{attribute 'linkalways'} 
{attribute 'no_explicit_call' := 'This FB is a CLASS and must be accessed using methods or properties'}
{attribute 'enable_dynamic_creation'}
FUNCTION_BLOCK _Array0to1OfARRAYTYP EXTENDS ArrayDatatypeBase
VAR CONSTANT
	lBound : DINT := 0;
	uBound : DINT := 1;
END_VAR
VAR
	localData : ARRAY [lBound..uBound] OF ARRAYTYP;
	activeData : REFERENCE TO ARRAY [lBound..uBound] OF ARRAYTYP REF= localData;
	elements : ARRAY [lBound..uBound] OF _ARRAYTYP();
	baseType : _ARRAYTYP();
END_VAR

PROPERTY PUBLIC Address : PVOID
GET
Address := ADR(activeData);
END_GET
END_PROPERTY

PROPERTY PUBLIC BaseDatatype : I_Datatype
GET
BaseDatatype := baseType;
END_GET
END_PROPERTY

METHOD PUBLIC ClearReference
VAR_INPUT
END_VAR
activeData REF= localData;
SetElementReference();
END_METHOD

METHOD PUBLIC Clone : I_Datatype
VAR
    pClone : POINTER TO _;
END_VAR
pClone := __NEW(_());
pClone^.Value := Value;
Clone := pClone^;
END_METHOD

METHOD FB_init : BOOL
VAR_INPUT
	bInitRetains : BOOL; // if TRUE, the retain variables are initialized (warm start / cold start)
	bInCopyCode : BOOL;  // if TRUE, the instance afterwards gets moved into the copy code (online change)
END_VAR
SetElementReference();
END_METHOD

METHOD PUBLIC GetElementAsDatatypeByIndex : I_Datatype
VAR_INPUT
	Index : DINT;
END_VAR
GetElementAsDatatypeByIndex := elements[Index];
END_METHOD

METHOD PUBLIC GetElementByIndex : REFERENCE TO _ARRAYTYP;
VAR_INPUT
	Index : DINT;
END_VAR
GetElementByIndex REF= elements[Index];
END_METHOD

PROPERTY PUBLIC LowerBound : DINT
GET
LowerBound := lBound;
END_GET
END_PROPERTY

METHOD PUBLIC MakeReferenceTo
VAR_INPUT
	ReferenceTarget : REFERENCE TO ARRAY [lBound..uBound] OF ARRAYTYP;
END_VAR
activeData REF= ReferenceTarget;
SetElementReference();
END_METHOD

METHOD PROTECTED OnSerializeArrayValues
VAR_INPUT
	Serializer : I_Serializer;
END_VAR
VAR
	i : DINT;
END_VAR
FOR i := lBound TO uBound DO
	elements[i].SerializeWith(Serializer);
END_FOR
END_METHOD

METHOD PROTECTED SetElementReference
VAR_INPUT
END_VAR
VAR
	i : DINT;
END_VAR
FOR i := lBound TO uBound DO
	elements[i].MakeReferenceTo(activeData[i]);
END_FOR
END_METHOD

PROPERTY PUBLIC Size : UDINT
GET
Size := SIZEOF(activeData);
END_GET
END_PROPERTY

METHOD PROTECTED TryDeserializeArrayValues : BOOL
VAR_INPUT
	Deserializer : I_Deserializer;
	Feedback : I_DeserializerFeedback;
END_VAR
VAR
	enumerator : I_DeserializerArrayForwardEnumerator;
	i : DINT;
END_VAR
enumerator := Deserializer.GetArrayEnumerator();
i := lBound;

WHILE enumerator.MoveNext() AND i <= uBound DO
	
	IF NOT elements[i].TryDeserializeFrom(enumerator.Current, Feedback) THEN
		EXIT;
	END_IF
	i := i + 1;

END_WHILE
enumerator.Dispose();
END_METHOD

METHOD TryMakeReferenceTo : BOOL
VAR_INPUT
	Target : I_Datatype;
END_VAR
VAR
	targetAsArray : I_ArrayDatatype;
	pTargetData : POINTER TO ARRAY [lBound..uBound] OF ARRAYTYP;
END_VAR
IF NOT Target.TryResolveAsArrayDatatype(targetAsArray) THEN
	RETURN;
END_IF

IF NOT (targetAsArray.Identifier = Identifier) THEN
	RETURN;
END_IF

pTargetData := Target.Address;
activeData REF= pTargetData^;
SetElementReference();
TryMakeReferenceTo := TRUE;
END_METHOD

PROPERTY PUBLIC UpperBound : DINT
GET
UpperBound := ubound;
END_GET
END_PROPERTY

PROPERTY PUBLIC Value : REFERENCE TO ARRAY [lBound..uBound] OF ARRAYTYP;
GET
Value ref= activeData;
END_GET
END_PROPERTY

END_FUNCTION_BLOCK

(* stored: Version 1.1.0.1, ProductVersion 3.1.4024.13
   POU _Array0to1OfARRAYTYP: Id {da1db718-2dc7-0680-1f34-420f519f6963}, SpecialFunc None
   Folder Core: Id {5c39afe2-7141-0130-2667-51939bb0c25d}
   Folder Constructor: Id {312294d5-c338-0e00-33ce-65fb362fadd9}
   Folder Protected: Id {35b6ee70-cbad-0432-1052-9e6c9f9aedba}
   Folder Customize: Id {f4f719dc-ac2c-0c9a-1b17-a2d5293b2885}
   Property Address: Id {107d8a18-5a85-07e8-0490-c9efdac61906}
   Get Get: Id {ced91096-f47d-0f6d-061c-7729ae761395}
   Property BaseDatatype: Id {d4f34257-75f1-0237-3bc9-14f6de04ea18}
   Get Get: Id {13c2eeee-719f-0bd5-235b-bd352bfe20d9}
   Method ClearReference: Id {33d83f31-ebc2-05e8-1d7d-7c6ebda0aad5}
   Method Clone: Id {bf1ddbe4-ab69-08e1-233f-f6370d208424}
   Method FB_init: Id {b1a23b05-0094-0813-36f0-0a76c62a99a8}
   Method GetElementAsDatatypeByIndex: Id {a25e9def-d2a5-09c2-1661-4577eb6bdbd5}
   Method GetElementByIndex: Id {05a8a4ae-936a-028b-34f7-ae8c32f6ddda}
   Property LowerBound: Id {4a60ccc3-0e38-0c8a-04bd-05ffd379d932}
   Get Get: Id {f837949f-80fb-0fa4-1ae8-a5355a97cd01}
   Method MakeReferenceTo: Id {7c2b7048-f4c9-00ff-1fdf-9dcc2ccfd7b9}
   Method OnSerializeArrayValues: Id {4048faae-cc77-0d91-14d3-5935f2b79a61}
   Method SetElementReference: Id {55ffa979-f6f1-0dc7-24de-49b96a58e601}
   Property Size: Id {a65b809b-acfd-04f8-04d4-a3000a28cb16}
   Get Get: Id {54b06454-092b-0b74-1483-257a36a4e94f}
   Method TryDeserializeArrayValues: Id {4711b22d-e75a-0be1-2ee2-db281762ff82}
   Method TryMakeReferenceTo: Id {6f67bda1-c408-03ef-329e-41da75f8b779}
   Property UpperBound: Id {5ded350d-81f1-0ddc-0a82-d9ebb7415312}
   Get Get: Id {0bda9718-b365-020f-3e73-118c4ba427ba}
   Property Value: Id {77a980b9-8441-045c-318a-7fb13eb11607}
   Get Get: Id {ca4d2820-0158-03df-1107-e7f1aa18ea05} *)
